TYPE ST_Modbus_Send_Frame :
STRUCT
	StartAddress		:WORD;
	sendQuantity		:WORD;
	SendData			:ARRAY [0..10] OF WORD;
END_STRUCT
END_TYPE

(* stored: Version 1.1.0.1
   DUT ST_Modbus_Send_Frame: Id {004d60f9-6d1e-4fe4-bacd-3597b6b8fdf9} *)
